FUNCTION_BLOCK itfSiloFlagsImplement IMPLEMENTS itfSiloFlags
VAR_INPUT
END_VAR
VAR_OUTPUT
END_VAR
VAR
	BufferedWeight : INT;
	TargetWeight : INT;
	LowProduct : BOOL;
END_VAR

PROPERTY pBufferedWeight : INT
GET
pBufferedWeight := BufferedWeight;
END_GET
SET
BufferedWeight := pBufferedWeight;
END_SET
END_PROPERTY

PROPERTY pLowProduct : BOOL
GET
pLowProduct := LowProduct;
END_GET
SET
LowProduct := pLowProduct;
END_SET
END_PROPERTY

PROPERTY pTargetWeight : INT
GET
pTargetWeight := TargetWeight;
END_GET
SET
TargetWeight := pTargetWeight;
END_SET
END_PROPERTY

END_FUNCTION_BLOCK

(* stored: Version 1.1.0.1, ProductVersion 3.1.4024.12
   POU itfSiloFlagsImplement: Id {af06416b-427c-4726-bd66-35bcaaba74aa}, SpecialFunc None
   Property pBufferedWeight: Id {4e254db4-469e-4979-8d38-bbc3faae0de8}
   Get Get: Id {d54c17c5-ee5d-495c-bfef-08e3ae8dee9b}
   Set Set: Id {025e1951-af4c-4ce0-8a16-89ff8429ec3d}
   Property pLowProduct: Id {045b3077-0c46-417a-853e-07c04eccd9ff}
   Get Get: Id {69a24c10-c685-4f76-b51a-0b92b9009b3b}
   Set Set: Id {8822b374-3d17-490f-946c-0774939e8909}
   Property pTargetWeight: Id {79142096-4691-4fd4-95ed-b86c4d44b986}
   Get Get: Id {bec8d8a7-dd59-424a-aaaa-6b5fdd9349dd}
   Set Set: Id {601e31e7-a6e0-47fa-b27f-9219ac54f66c} *)
